// LS Electric XG5000 project: 과년70_2
// PLC NewPLC
// module base 0 slot 0: 입출력 모듈:XBC-DR20S (DC 24V 입력 12점, 릴레이 출력 8점)

PROGRAM NewProgram (task: 스캔 프로그램)

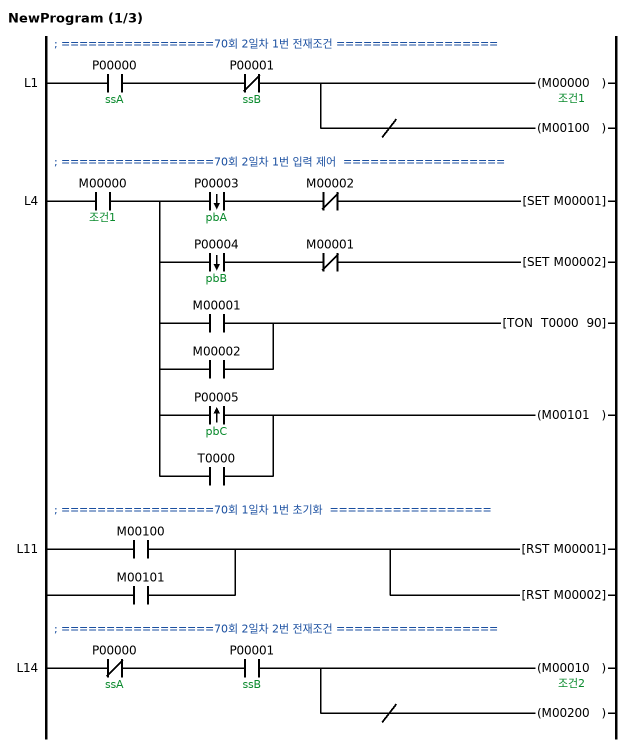
// =================70회 2일차 1번 전재조건 ==================
; L1
LOAD      P00000	// ssA
AND NOT   P00001	// ssB
OUT       M00000	// 조건1
NOT
OUT       M00100
// =================70회 2일차 1번 입력 제어  ==================
; L4
LOAD      M00000	// 조건1
MPUSH
ANDN      P00003	// pbA
AND NOT   M00002
SET       M00001
MLOAD
ANDN      P00004	// pbB
AND NOT   M00001
SET       M00002
MLOAD
LOAD      M00001
OR        M00002
AND LOAD
TON       T0000 90
MPOP
LOADP     P00005	// pbC
OR        T0000
AND LOAD
OUT       M00101
// =================70회 1일차 1번 초기화  ==================
; L11
LOAD      M00100
OR        M00101
RST       M00001
RST       M00002
// =================70회 2일차 2번 전재조건 ==================
; L14
LOAD NOT  P00000	// ssA
AND       P00001	// ssB
OUT       M00010	// 조건2
NOT
OUT       M00200

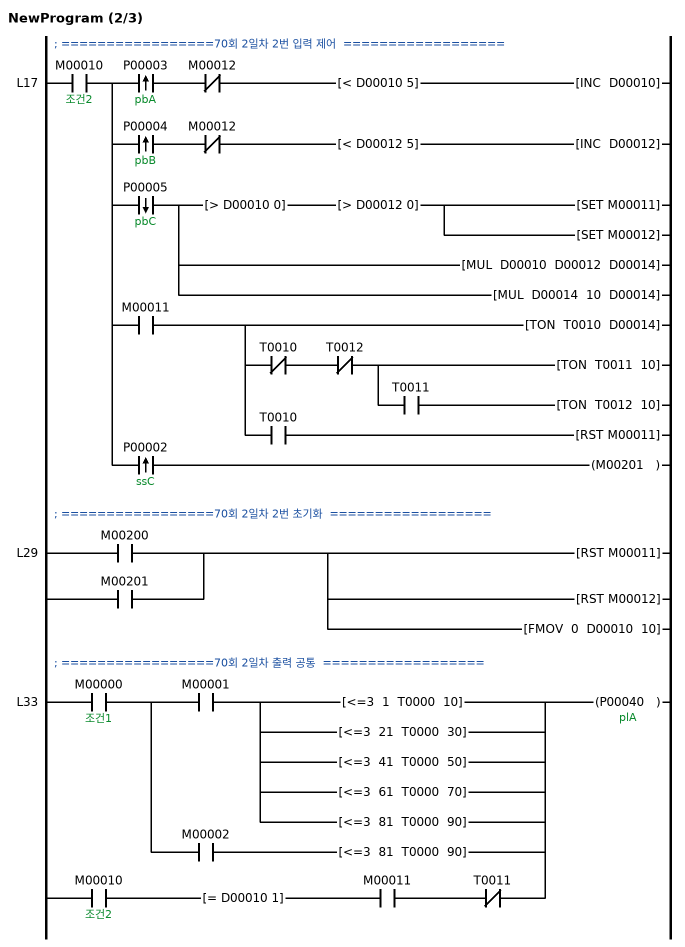
// =================70회 2일차 2번 입력 제어  ==================
; L17
LOAD      M00010	// 조건2
MPUSH
ANDP      P00003	// pbA
AND NOT   M00012
AND<      D00010 5
INC       D00010
MLOAD
ANDP      P00004	// pbB
AND NOT   M00012
AND<      D00012 5
INC       D00012
MLOAD
ANDN      P00005	// pbC
MPUSH
AND>      D00010 0
AND>      D00012 0
SET       M00011
SET       M00012
MPOP
MUL       D00010 D00012 D00014
MUL       D00014 10 D00014
MLOAD
AND       M00011
TON       T0010 D00014
MPUSH
AND NOT   T0010
AND NOT   T0012
TON       T0011 10
AND       T0011
TON       T0012 10
MPOP
AND       T0010
RST       M00011
MPOP
ANDP      P00002	// ssC
OUT       M00201
// =================70회 2일차 2번 초기화  ==================
; L29
LOAD      M00200
OR        M00201
RST       M00011
RST       M00012
FMOV      0 D00010 10
// =================70회 2일차 출력 공통  ==================
; L33
LOAD      M00000	// 조건1
LOAD      M00001
LOAD<=3   1 T0000 10
OR<=3     21 T0000 30
OR<=3     41 T0000 50
OR<=3     61 T0000 70
OR<=3     81 T0000 90
AND LOAD
LOAD      M00002
AND<=3    81 T0000 90
OR LOAD
AND LOAD
LOAD      M00010	// 조건2
AND=      D00010 1
AND       M00011
AND NOT   T0011
OR LOAD
OUT       P00040	// plA

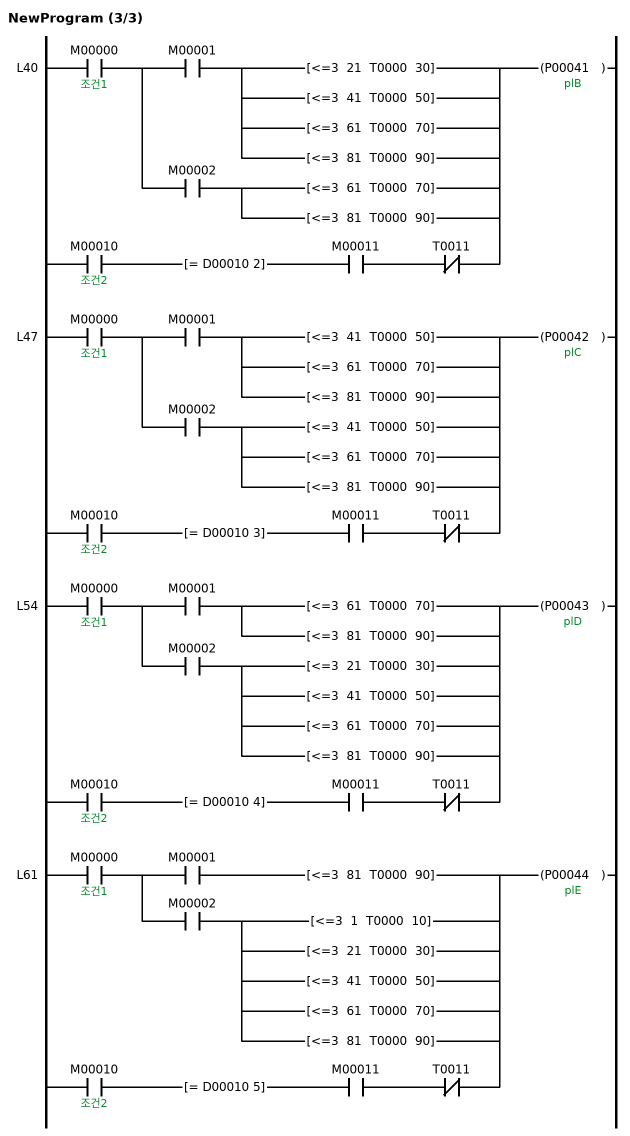
; L40
LOAD      M00000	// 조건1
LOAD      M00001
LOAD<=3   21 T0000 30
OR<=3     41 T0000 50
OR<=3     61 T0000 70
OR<=3     81 T0000 90
AND LOAD
LOAD      M00002
LOAD<=3   61 T0000 70
OR<=3     81 T0000 90
AND LOAD
OR LOAD
AND LOAD
LOAD      M00010	// 조건2
AND=      D00010 2
AND       M00011
AND NOT   T0011
OR LOAD
OUT       P00041	// plB
; L47
LOAD      M00000	// 조건1
LOAD      M00001
LOAD<=3   41 T0000 50
OR<=3     61 T0000 70
OR<=3     81 T0000 90
AND LOAD
LOAD      M00002
LOAD<=3   41 T0000 50
OR<=3     61 T0000 70
OR<=3     81 T0000 90
AND LOAD
OR LOAD
AND LOAD
LOAD      M00010	// 조건2
AND=      D00010 3
AND       M00011
AND NOT   T0011
OR LOAD
OUT       P00042	// plC
; L54
LOAD      M00000	// 조건1
LOAD      M00001
LOAD<=3   61 T0000 70
OR<=3     81 T0000 90
AND LOAD
LOAD      M00002
LOAD<=3   21 T0000 30
OR<=3     41 T0000 50
OR<=3     61 T0000 70
OR<=3     81 T0000 90
AND LOAD
OR LOAD
AND LOAD
LOAD      M00010	// 조건2
AND=      D00010 4
AND       M00011
AND NOT   T0011
OR LOAD
OUT       P00043	// plD
; L61
LOAD      M00000	// 조건1
LOAD      M00001
AND<=3    81 T0000 90
LOAD      M00002
LOAD<=3   1 T0000 10
OR<=3     21 T0000 30
OR<=3     41 T0000 50
OR<=3     61 T0000 70
OR<=3     81 T0000 90
AND LOAD
OR LOAD
AND LOAD
LOAD      M00010	// 조건2
AND=      D00010 5
AND       M00011
AND NOT   T0011
OR LOAD
OUT       P00044	// plE